FUNCTION_BLOCK xscal
VAR_INPUT
    b_n: DINT;
    a: LREAL;
    ix0: DINT;
END_VAR
VAR_IN_OUT
    x: ARRAY [0..29] OF LREAL;
END_VAR
VAR_TEMP
    b: DINT;
    k: DINT;
END_VAR

b := (ix0 + b_n) - 1;
k := ix0;
WHILE k <= b DO
    x[k - 1] := x[k - 1] * a;
    k := k + 1;
END_WHILE;

END_FUNCTION_BLOCK

(* stored: Version 1.1.0.1, ProductVersion 3.1.4024.12
   POU xscal: Id {bfd09ec0-f8de-424d-af91-988a3b3465d0}, SpecialFunc None *)
